TYPE ST_IOT_SentStateLog :
STRUCT
	bUpdate			: BOOL;
	bMessageSent	: BOOL;
	LastIndexSent	: INT;
	LastIndex		: INT;
END_STRUCT
END_TYPE

(* stored: Version 1.1.0.1, ProductVersion 3.1.4026.18
   DUT ST_IOT_SentStateLog: Id {32701801-f332-4954-8717-1fe3a567d283} *)
